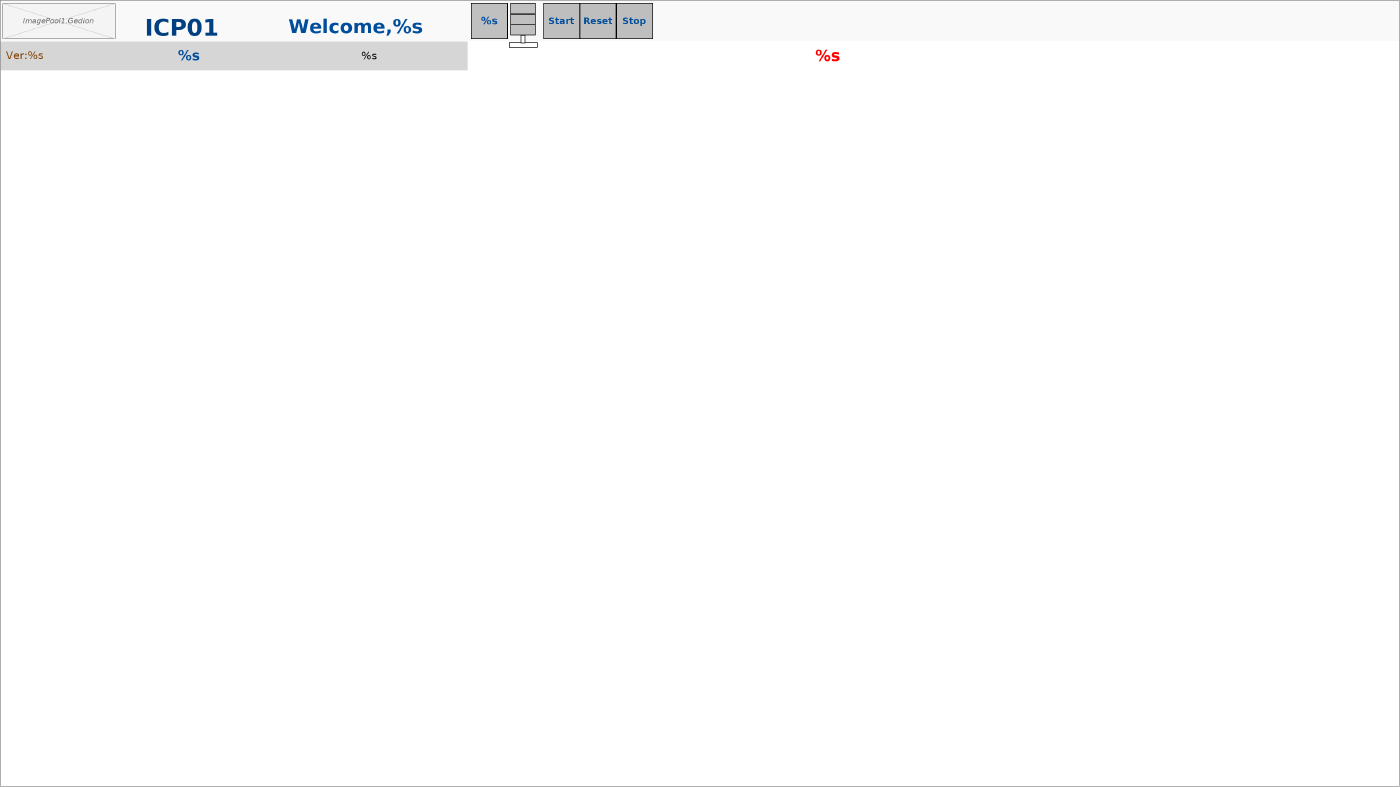
VISUALIZATION MainFrame  // 1920x1080, background image ImagePool1.background
VAR_IN_OUT
	userData:MainFram;
END_VAR
    Rectangle (0,57 641x39)
    Rectangle (373,57 267x39), "%s", text variable: userData.ShowTime
    Rectangle (646,57 979x39), "%s", text variable: userData.ErrWTxtShow, invisible if: Not (gRunningState=RunningStatus.eErrorState)
    Rectangle (5,57 142x38), "Ver:%s", text variable: userData.versions
    Rectangle (0,0 1920x56)
    InvisibleInput (0,0 1x12)
    InvisibleInput (0,0 1x1)
    Rectangle (363,20 250x33), "Welcome,%s", text variable: gCurrentUser
    Image (3,4 155x49), image: ImagePool1.Gedion
    Rectangle (173,23 175x30), "ICP01"
    Group (698,4 45x49)
        Rectangle (2,0 34x15), colour toggle: userData.RedLamp
        Rectangle (2,15 34x15), colour toggle: userData.YellowLamp
        Rectangle (2,29 34x15), colour toggle: userData.GreenLamp
        Rectangle (0,54 39x7)
        Rectangle (16,44 6x11)
    Rectangle (745,4 50x49), "Start", colour toggle: userData.StartLamp
        tap userData.Start
    Rectangle (795,4 50x49), "Reset", colour toggle: userData.ResetLamp
        tap userData.Reset
    Rectangle (845,4 50x49), "Stop", colour toggle: userData.StopLamp
        tap userData.Stop
    Rectangle (646,4 50x49), "%s", tooltip "A:Auto Running E:Error Running H:Homing M:Manual Running P:Pause Running S:Stop Running", text variable: userData.RunStateTxt
    Rectangle (153,57 213x39), "%s", text variable: fbMachineState.RunStateTxt
END_VISUALIZATION

(* stored: Version 1.1.0.1, ProductVersion 3.1.4024.12
   Visu MainFrame: Id {5a8a8dd3-0247-47f3-aaee-7cbe0aedbf7e} *)
